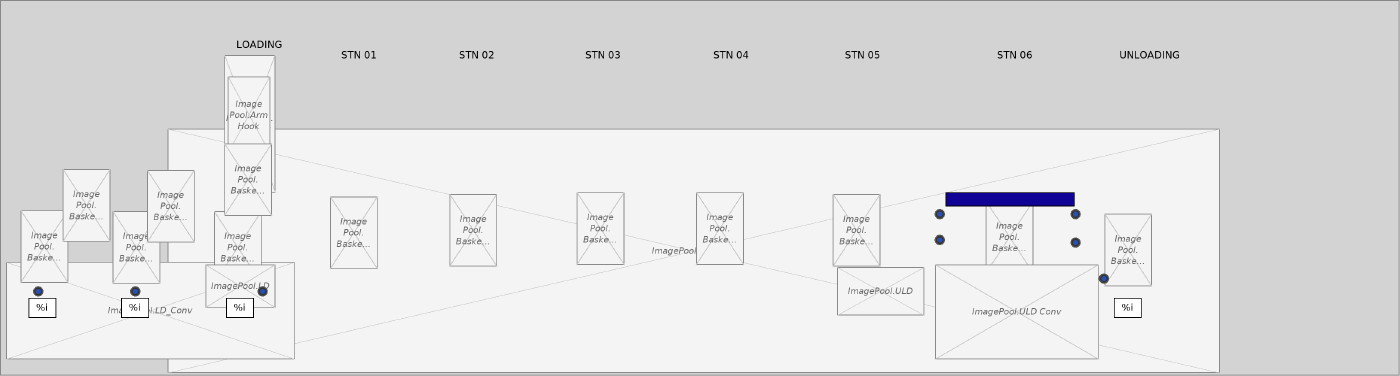
VISUALIZATION Popup_Machine_Manual  // 1629x438
    Rectangle (0,0 1629x438)
    Image (195,150 1224x284), image: ImagePool.Machine
    Label (378,44 80x40), "STN 01"
    Label (515,44 80x40), "STN 02"
    Label (662,44 80x40), "STN 03"
    Label (811,44 80x40), "STN 04"
    Label (964,44 80x40), "STN 05"
    Label (1141,44 80x40), "STN 06"
    Label (251,32 102x40), "LOADING"
    Label (1285,44 106x40), "UNLOADING"
    Group (384,229 55x84)
        Image (0,0 55x84), invisible if: NOT.ARbBasketBdFlag[2], image: ImagePool.Basket Red
            OnMouseDown: execute { DSStnBasketInfo[1].iProductRecipeNo:=0; }
        Image (0,0 55x84), invisible if: NOT.ARbBasketGdFlag[2], image: ImagePool.Basket Green
            OnMouseDown: execute { DSStnBasketInfo[1].iProductRecipeNo:=0; }
    Group (523,226 55x84)
        Image (0,0 55x84), invisible if: NOT.ARbBasketBdFlag[3], image: ImagePool.Basket Red
            OnMouseDown: execute { DSStnBasketInfo[2].iProductRecipeNo:=0; }
        Image (0,0 55x84), invisible if: NOT.ARbBasketGdFlag[3], image: ImagePool.Basket Green
            OnMouseDown: execute { DSStnBasketInfo[2].iProductRecipeNo:=0; }
    Group (671,224 55x84)
        Image (0,0 55x84), invisible if: NOT.ARbBasketBdFlag[4], image: ImagePool.Basket Red
            OnMouseDown: execute { DSStnBasketInfo[3].iProductRecipeNo:=0; }
        Image (0,0 55x84), invisible if: NOT.ARbBasketGdFlag[4], image: ImagePool.Basket Green
            OnMouseDown: execute { DSStnBasketInfo[3].iProductRecipeNo:=0; }
    Group (810,224 55x84)
        Image (0,0 55x84), invisible if: NOT.ARbBasketBdFlag[5], image: ImagePool.Basket Red
            OnMouseDown: execute { DSStnBasketInfo[4].iProductRecipeNo:=0; }
        Image (0,0 55x84), invisible if: NOT.ARbBasketGdFlag[5], image: ImagePool.Basket Green
            OnMouseDown: execute { DSStnBasketInfo[4].iProductRecipeNo:=0; }
    Group (969,226 55x84)
        Image (0,0 55x84), invisible if: NOT.ARbBasketBdFlag[6], image: ImagePool.Basket Red
            OnMouseDown: execute { DSStnBasketInfo[5].iProductRecipeNo:=0; }
        Image (0,0 55x84), invisible if: NOT.ARbBasketGdFlag[6], image: ImagePool.Basket Green
            OnMouseDown: execute { DSStnBasketInfo[5].iProductRecipeNo:=0; }
    Group (1147,234 55x84)
        Image (0,0 55x84), invisible if: NOT.ARbBasketBdFlag[7], image: ImagePool.Basket Red
            OnMouseDown: execute { DSStnBasketInfo[6].iProductRecipeNo:=0; }
        Image (0,0 55x84), invisible if: NOT.ARbBasketGdFlag[7], image: ImagePool.Basket Green
            OnMouseDown: execute { DSStnBasketInfo[6].iProductRecipeNo:=0; }
    Image (7,305 336x113), image: ImagePool.LD_Conv
    Image (249,246 55x84), invisible if: NOT.ARbBasketGdFlag[1], image: ImagePool.Basket Green
        OnMouseDown: execute { AR2sDSCv_LdConfirmBasketInfo[1,3].iProductRecipeNo:=0; }
    Image (24,245 55x84), invisible if: NOT AR2sDSCv_LdConfirmBasketInfo[1,1].bAvailibility, image: ImagePool.Basket Green
        OnMouseDown: execute { AR2sDSCv_LdConfirmBasketInfo[1,1].iProductRecipeNo:=0; }
    Image (239,308 81x50), image: ImagePool.LD
    Image (261,64 59x160), text variable: DSArmBasketInfo[1].iProductRecipeNo, image: ImagePool.Arm Body
        p3560616238: HMI_Function.MotionX
        OnMouseDown: write the text variable via VisuDialogs.Numpad
    Image (265,89 49x90), text variable: DSArmBasketInfo[1].iProductRecipeNo, image: ImagePool.Arm Hook
        p3560616238: HMI_Function.MotionX
        p2738717112: HMI_Function.MotionY
        OnMouseDown: write the text variable via VisuDialogs.Numpad
    Image (261,167 55x84), invisible if: NOT.ARbBasketBdFlag[16], image: ImagePool.Basket Red
        p3560616238: HMI_Function.MotionX
        p2738717112: HMI_Function.MotionY
        OnMouseDown: execute { DSArmBasketInfo[1].iProductRecipeNo:=0; }
    Image (261,167 55x84), invisible if: NOT.ARbBasketGdFlag[16], image: ImagePool.Basket Green
        p2738717112: HMI_Function.MotionY
        p3560616238: HMI_Function.MotionX
        OnMouseDown: execute { DSArmBasketInfo[1].iProductRecipeNo:=0; }
    Image (974,311 101x56), image: ImagePool.ULD
    Image (131,246 55x84), invisible if: NOT AR2sDSCv_LdConfirmBasketInfo[1,2].bAvailibility, image: ImagePool.Basket Green
        OnMouseDown: execute { AR2sDSCv_LdConfirmBasketInfo[1,2].iProductRecipeNo:=0; }
    Image (73,197 55x84), invisible if: NOT AR2sDSCv_LdTransferBasketInfo[1,1].bAvailibility, image: ImagePool.Basket Blue
        OnMouseDown: execute { AR2sDSCv_LdTransferBasketInfo[1,1].iProductRecipeNo:=0; }
    Image (171,198 55x84), invisible if: NOT AR2sDSCv_LdTransferBasketInfo[1,2].bAvailibility, image: ImagePool.Basket Blue
        OnMouseDown: execute { AR2sDSCv_LdTransferBasketInfo[1,2].iProductRecipeNo:=0;; }
    Image (1285,249 55x84), invisible if: NOT.ARbBasketBdFlag[12], image: ImagePool.Basket Red
        OnMouseDown: execute { AR2sDSCv_UldConfirmBasketInfo[1,1].iProductRecipeNo:=0; }
    Image (1285,249 55x84), invisible if: NOT.ARbBasketGdFlag[12], image: ImagePool.Basket Green
        OnMouseDown: execute { AR2sDSCv_UldConfirmBasketInfo[1,1].iProductRecipeNo:=0; }
    Image (1088,308 190x110), image: ImagePool.ULD Conv
    Lamp1 (1278,318 13x13), variable: ARbDI[eX12011_UnloadingSensor_BasketDetection], style: Lamp-Lamp1-Blue
    Rectangle (1296,347 32x23), "%i", text variable: AR2sDSCv_UldConfirmBasketInfo[1,1].iProductRecipeNo
        OnMouseDown: write the text variable via VisuDialogs.Numpad
    Rectangle (263,347 32x23), "%i", text variable: AR2sDSCv_LdConfirmBasketInfo[1,3].iProductRecipeNo
        OnMouseDown: write the text variable via VisuDialogs.Numpad
    Rectangle (141,347 32x23), "%i", text variable: AR2sDSCv_LdConfirmBasketInfo[1,2].iProductRecipeNo
        OnMouseDown: write the text variable via VisuDialogs.Numpad
    Rectangle (33,347 32x23), "%i", text variable: AR2sDSCv_LdConfirmBasketInfo[1,1].iProductRecipeNo
        OnMouseDown: write the text variable via VisuDialogs.Numpad
    Lamp1 (299,333 13x13), variable: ARbDI[eX13002_LoadingConveyorSensor_Pick], style: Lamp-Lamp1-Blue
    Lamp1 (38,333 13x13), variable: ARbDI[eX13000_LoadingConveyorSensor_Feed], style: Lamp-Lamp1-Blue
    Lamp1 (151,333 13x13), variable: ARbDI[eX13001_LoadingConveyorSensor_Index], style: Lamp-Lamp1-Blue
    Lamp1 (1087,243 13x13), variable: ARbDI[eX12101_Stn06SlidingDoorRs01_Unclamp], style: Lamp-Lamp1-Blue
    Lamp1 (1087,273 13x13), variable: ARbDI[eX12100_Stn06SlidingDoorRs01_Clamp], style: Lamp-Lamp1-Blue
    Lamp1 (1245,276 13x13), variable: ARbDI[eX12102_Stn06SlidingDoorRs02_Clamp], style: Lamp-Lamp1-Blue
    Lamp1 (1245,243 13x13), variable: ARbDI[eX12103_Stn06SlidingDoorRs02_Unclamp], style: Lamp-Lamp1-Blue
    Rectangle (1100,224 150x16), invisible if: NOT ARbDI[eX12008_Stn06SlidingDoorRs_Close]
END_VISUALIZATION

(* stored: Version 1.1.0.1, ProductVersion 3.1.4024.12
   Visu Popup_Machine_Manual: Id {71aa11d1-9dd0-4c61-9726-5bedaac0ff8a} *)
